(* PLC project MXEN3002 sorting, MXEN3002 Festo Station Control 1.0 *)
(* stored: creationDateTime 2026-07-20T16:20:05 *)

FUNCTION_BLOCK FB_Panel
  VAR_INPUT
    s1_start : BOOL;
    s2_stop : BOOL;
    s4_reset : BOOL;
    error_in : BOOL;
    reset_done : BOOL;
  END_VAR
  VAR_OUTPUT
    run_mode : BOOL;
    reset_mode : BOOL;
    pause_mode : BOOL;
    error_mode : BOOL;
    start_light : BOOL;
    reset_light : BOOL;
  END_VAR
  VAR
    reset_mode : BOOL;
    pause_mode : BOOL;
    error_mode : BOOL;
    start_light : BOOL;
    reset_light : BOOL;
    state : INT := 0;
  END_VAR

IF error_in AND state <> 3 THEN
    state := 3;                          // ERROR forced from any state
ELSIF state = 0 THEN                     // PAUSE
    IF s1_start THEN
        state := 1;
    ELSIF s4_reset THEN
        state := 2;
    END_IF;
ELSIF state = 1 THEN                     // RUN
    IF s2_stop THEN state := 0; END_IF;  // S4 ignored here
ELSIF state = 2 THEN                     // RESET
    IF s2_stop OR reset_done THEN state := 0; END_IF;   // S1 ignored here
ELSIF state = 3 THEN                     // ERROR
    IF s4_reset THEN state := 2; END_IF; // clears fault, begins reset/homing
END_IF;

run_mode    := (state = 1);
pause_mode  := (state = 0);
reset_mode  := (state = 2);
error_mode  := (state = 3);
start_light := run_mode;
reset_light := reset_mode;
END_FUNCTION_BLOCK

FUNCTION_BLOCK FB_Actuator_T2
  VAR_INPUT
    run_mode : BOOL;
    pause_mode : BOOL;
    reset_mode : BOOL;
    error_mode : BOOL;
    sensor_home : BOOL;
    sensor_end : BOOL;
    go : BOOL;
    t_stall : TIME := T#2s;
    robust : BOOL := FALSE;
  END_VAR
  VAR_OUTPUT
    at_home : BOOL;
    to_end : BOOL;
    at_end : BOOL;
    to_home : BOOL;
    valve_extend : BOOL;
    error : BOOL;
  END_VAR
  VAR
    to_end : BOOL;
    at_end : BOOL;
    to_home : BOOL;
    valve_extend : BOOL;
    error : BOOL;
    state : INT := 0;
    stall : TON;
    moving : BOOL;
  END_VAR

CASE state OF
0:  (* AT_HOME *)
    IF error_mode THEN state := 4;
    ELSIF reset_mode THEN
        IF NOT sensor_home THEN state := 3; END_IF;
    ELSIF run_mode AND go THEN state := 1;
    END_IF;
1:  (* TO_END -- stroke completes regardless of pause *)
    IF error_mode THEN state := 4;
    ELSIF sensor_end THEN state := 2;
    END_IF;
2:  (* AT_END -- valve held extended; only run advances to retract *)
    IF error_mode THEN state := 4;
    ELSIF reset_mode THEN state := 3;
    ELSIF run_mode THEN state := 3;
    END_IF;
3:  (* TO_HOME -- valve off, spring retracts, completes regardless of pause *)
    IF error_mode THEN state := 4;
    ELSIF sensor_home THEN state := 0;
    END_IF;
4:  (* ERROR *)
    IF reset_mode THEN
        IF sensor_home THEN state := 0; ELSE state := 3; END_IF;
    END_IF;
END_CASE;

valve_extend := (state = 1) OR (state = 2);
IF state = 4 THEN valve_extend := FALSE; END_IF;

moving := (state = 1) OR (state = 3);
stall(IN := robust AND moving, PT := t_stall);
IF stall.Q THEN
    state := 4;
    valve_extend := FALSE;
END_IF;

at_home := (state = 0);
to_end  := (state = 1);
at_end  := (state = 2);
to_home := (state = 3);
error   := (state = 4);
END_FUNCTION_BLOCK

FUNCTION_BLOCK FB_Actuator_T3
  VAR_INPUT
    run_mode : BOOL;
    pause_mode : BOOL;
    reset_mode : BOOL;
    error_mode : BOOL;
    sensor_home : BOOL;
    go : BOOL;
    t_stroke : TIME := T#1s;
    t_stall : TIME := T#2s;
    robust : BOOL := FALSE;
  END_VAR
  VAR_OUTPUT
    at_home : BOOL;
    to_end : BOOL;
    at_end : BOOL;
    to_home : BOOL;
    valve_extend : BOOL;
    error : BOOL;
  END_VAR
  VAR
    to_end : BOOL;
    at_end : BOOL;
    to_home : BOOL;
    valve_extend : BOOL;
    error : BOOL;
    state : INT := 0;
    strokeT : TON;
    stallT : TON;
  END_VAR

CASE state OF
0:  (* AT_HOME *)
    IF error_mode THEN state := 4;
    ELSIF reset_mode THEN
        IF NOT sensor_home THEN state := 3; END_IF;
    ELSIF run_mode AND go THEN state := 1;
    END_IF;
1:  (* TO_END -- no sensor, trust the stroke timer *)
    IF error_mode THEN state := 4;
    ELSIF strokeT.Q THEN state := 2;
    END_IF;
2:  (* AT_END *)
    IF error_mode THEN state := 4;
    ELSIF reset_mode THEN state := 3;
    ELSIF run_mode THEN state := 3;
    END_IF;
3:  (* TO_HOME -- retract, sensor_home ends it *)
    IF error_mode THEN state := 4;
    ELSIF sensor_home THEN state := 0;
    END_IF;
4:  (* ERROR *)
    IF reset_mode THEN
        IF sensor_home THEN state := 0; ELSE state := 3; END_IF;
    END_IF;
END_CASE;

valve_extend := (state = 1) OR (state = 2);
IF state = 4 THEN valve_extend := FALSE; END_IF;

strokeT(IN := (state = 1), PT := t_stroke);
stallT (IN := robust AND (state = 3), PT := t_stall);   // retract-only stall
IF stallT.Q THEN
    state := 4;
    valve_extend := FALSE;
END_IF;

at_home := (state = 0);
to_end  := (state = 1);
at_end  := (state = 2);
to_home := (state = 3);
error   := (state = 4);
END_FUNCTION_BLOCK

PROGRAM Main_Sorting
  VAR
    Panel : FB_Panel;
    Branch1 : FB_Actuator_T2;
    Branch2 : FB_Actuator_T2;
    Stopper : FB_Actuator_T3;
    pos : INT := 0;
    dest : INT := 0;
    have : BOOL;
    ROBUST : BOOL := TRUE;
    CAP : INT := 5;
  END_VAR

reset_done := Branch1.at_home AND Branch2.at_home;
Panel(s1_start := Panel_S1, s2_stop := Panel_S2, s4_reset := Panel_S4,
      error_in := fault, reset_done := reset_done);

IF Panel.reset_mode OR Panel.error_mode THEN
    have := FALSE; pos := 0;
END_IF;

slide_full := Station_B4 OR (s1c >= CAP) OR (s2c >= CAP) OR (s3c >= CAP);

conveyor := FALSE; go_b1 := FALSE; go_b2 := FALSE; go_stop := FALSE;
IF Panel.run_mode AND NOT slide_full THEN
    IF NOT have THEN
        IF Part_AV THEN                        // classify newly released piece
            metal := Station_B2;
            black := NOT Station_B3;
            red   := Station_B3 AND NOT Station_B2;
            IF metal THEN dest := 0;
            ELSIF red THEN dest := 1;
            ELSE dest := 2; END_IF;
            have := TRUE; pos := 0;
            go_stop := TRUE;                   // pulse stopper to admit the piece
        END_IF;
    ELSE
        CASE dest OF
        0:  (* branch 1 *)
            IF pos < 1 THEN conveyor := TRUE; pos := pos + 1;
            ELSE
                go_b1 := TRUE;
                IF Branch1.at_end THEN s1c := s1c + 1; have := FALSE; END_IF;
            END_IF;
        1:  (* branch 2 *)
            IF pos < 2 THEN conveyor := TRUE; pos := pos + 1;
            ELSE
                go_b2 := TRUE;
                IF Branch2.at_end THEN s2c := s2c + 1; have := FALSE; END_IF;
            END_IF;
        2:  (* straight through to end slide *)
            IF pos < 3 THEN conveyor := TRUE; pos := pos + 1;
            ELSE s3c := s3c + 1; have := FALSE; END_IF;
        END_CASE;
    END_IF;
END_IF;

Branch1(run_mode := Panel.run_mode, pause_mode := Panel.pause_mode,
    reset_mode := Panel.reset_mode, error_mode := Panel.error_mode,
    sensor_home := Station_1B1, sensor_end := Station_1B2, go := go_b1,
    t_stall := T#2s, robust := ROBUST);

Branch2(run_mode := Panel.run_mode, pause_mode := Panel.pause_mode,
    reset_mode := Panel.reset_mode, error_mode := Panel.error_mode,
    sensor_home := Station_2B1, sensor_end := Station_2B2, go := go_b2,
    t_stall := T#2s, robust := ROBUST);

Stopper(run_mode := Panel.run_mode, pause_mode := Panel.pause_mode,
    reset_mode := Panel.reset_mode, error_mode := Panel.error_mode,
    sensor_home := TRUE, go := go_stop,
    t_stroke := T#1s, t_stall := T#2s, robust := ROBUST);

// Robust faults (3.2): a branch stalled/held, or any slide full. Piece-removed
// (a piece taken off the conveyor before a slide) is inferred as: routing a
// piece but Part_AV lost mid-line -- VERIFY sensor behaviour on the bench.
fault := (ROBUST AND (Branch1.error OR Branch2.error))
    OR (Panel.run_mode AND slide_full)
    OR (ROBUST AND Panel.run_mode AND have AND pos >= 1 AND NOT Part_AV);

// ---- physical outputs ----
Station_K1  := conveyor AND NOT Panel.error_mode;   // Conveyor Motor ON
Station_1Y1 := Branch1.valve_extend;                // Branch 1 extend
Station_2Y1 := Branch2.valve_extend;                // Branch 2 extend
Station_3Y1 := Stopper.valve_extend;                // Stopper retract (release)
Station_H1  := Panel.start_light;
Station_H2  := Panel.reset_light;
Station_H3  := slide_full;                          // Q1
Station_H4  := Panel.error_mode;                    // Q2
IP_N_FO     := Panel.run_mode;                      // station occupied
END_PROGRAM

CONFIGURATION Config0
  RESOURCE Resource0 ON PLC
    VAR_GLOBAL
      Part_AV AT %IX0.00 : BOOL;  (* Workpiece Available *)
      Station_B2 AT %IX0.01 : BOOL;  (* Metallic Workpiece *)
      Station_B3 AT %IX0.02 : BOOL;  (* Workpiece not black *)
      Station_B4 AT %IX0.03 : BOOL;  (* Slide Full *)
      Station_1B1 AT %IX0.04 : BOOL;  (* Branch 1 Retracted (T2 sensor_home) *)
      Station_1B2 AT %IX0.05 : BOOL;  (* Branch 1 Extended (T2 sensor_end) *)
      Station_2B1 AT %IX0.06 : BOOL;  (* Branch 2 Retracted (T2 sensor_home) *)
      Station_2B2 AT %IX0.07 : BOOL;  (* Branch 2 Extended (T2 sensor_end) *)
      Panel_S1 AT %IX0.08 : BOOL;  (* Start Button *)
      Panel_S2 AT %IX0.09 : BOOL;  (* Stop Button *)
      Panel_S4 AT %IX0.11 : BOOL;  (* Reset Button *)
      Station_K1 AT %QX1.00 : BOOL;  (* Conveyor Motor ON *)
      Station_1Y1 AT %QX1.01 : BOOL;  (* Branch 1 to extend (T2 valve_extend) *)
      Station_2Y1 AT %QX1.02 : BOOL;  (* Branch 2 to extend (T2 valve_extend) *)
      Station_3Y1 AT %QX1.03 : BOOL;  (* Stopper to Retract (T3 valve_extend) *)
      IP_N_FO AT %QX1.07 : BOOL;  (* Station Occupied *)
      Station_H1 AT %QX1.08 : BOOL;  (* Start Indicator Light *)
      Station_H2 AT %QX1.09 : BOOL;  (* Reset Indicator Light *)
      Station_H3 AT %QX1.10 : BOOL;  (* Q1 indicator light *)
      Station_H4 AT %QX1.11 : BOOL;  (* Q2 indicator light *)
    END_VAR
    TASK PrimaryTask(INTERVAL := T#10ms, PRIORITY := 0);
    PROGRAM Main_Sorting_inst WITH PrimaryTask : Main_Sorting;
  END_RESOURCE
END_CONFIGURATION
